// TIA Portal V17 export
// export: Created 2025-03-07T09:24:30.3982886Z, ExportSetting WithDefaults, DisplayName Totally Integrated Automation Portal, DisplayVersion V17 Update 8, DisplayName TIA Portal Openness, DisplayVersion V17 Update 8, DisplayName TIA Portal Version Control Interface, DisplayVersion V17, DisplayName SINAMICS Startdrive Advanced, DisplayVersion V17 SP2, DisplayName SINAMICS Startdrive G110M, G120, G120C, G120D, G120P, G115D, DisplayVersion V17 SP2, DisplayName SINAMICS Startdrive G130, G150, S120, S150, SINAMICS MV, S210, DisplayVersion V17 SP2, DisplayName STEP 7 Professional, DisplayVersion V17 Update 8, DisplayName SINUMERIK ONE STEP 7 Toolbox, DisplayVersion V17 Update 12, DisplayName SINUMERIK 840D sl STEP 7 Toolbox, DisplayVersion V17 Update 12, DisplayName STEP 7 Safety, DisplayVersion V17 Update 6, DisplayName WinCC Advanced, DisplayVersion V17 Update 8
FUNCTION "FC2202_PROFINET" : Void   // FC2202, LAD
{ S7_Optimized_Access := 'FALSE' }
AUTHOR : ETXETAR
VERSION : 1.0
// stored: AutoNumber false, IsIECCheckEnabled false, SetENOAutomatically false, UDAEnableTagReadback false
   VAR_TEMP
      COMMAND : Int;   // COMMAND
      BUSY : Bool;   // BUSY
   END_VAR
   VAR CONSTANT
      FC_NUMBER : Int := 2202;
   END_VAR
   VAR_TEMP   // added for the SCL form of the ladder/FBD networks
      _w1 : Bool;
   END_VAR
BEGIN

REGION Network 1: DEVICES STATES
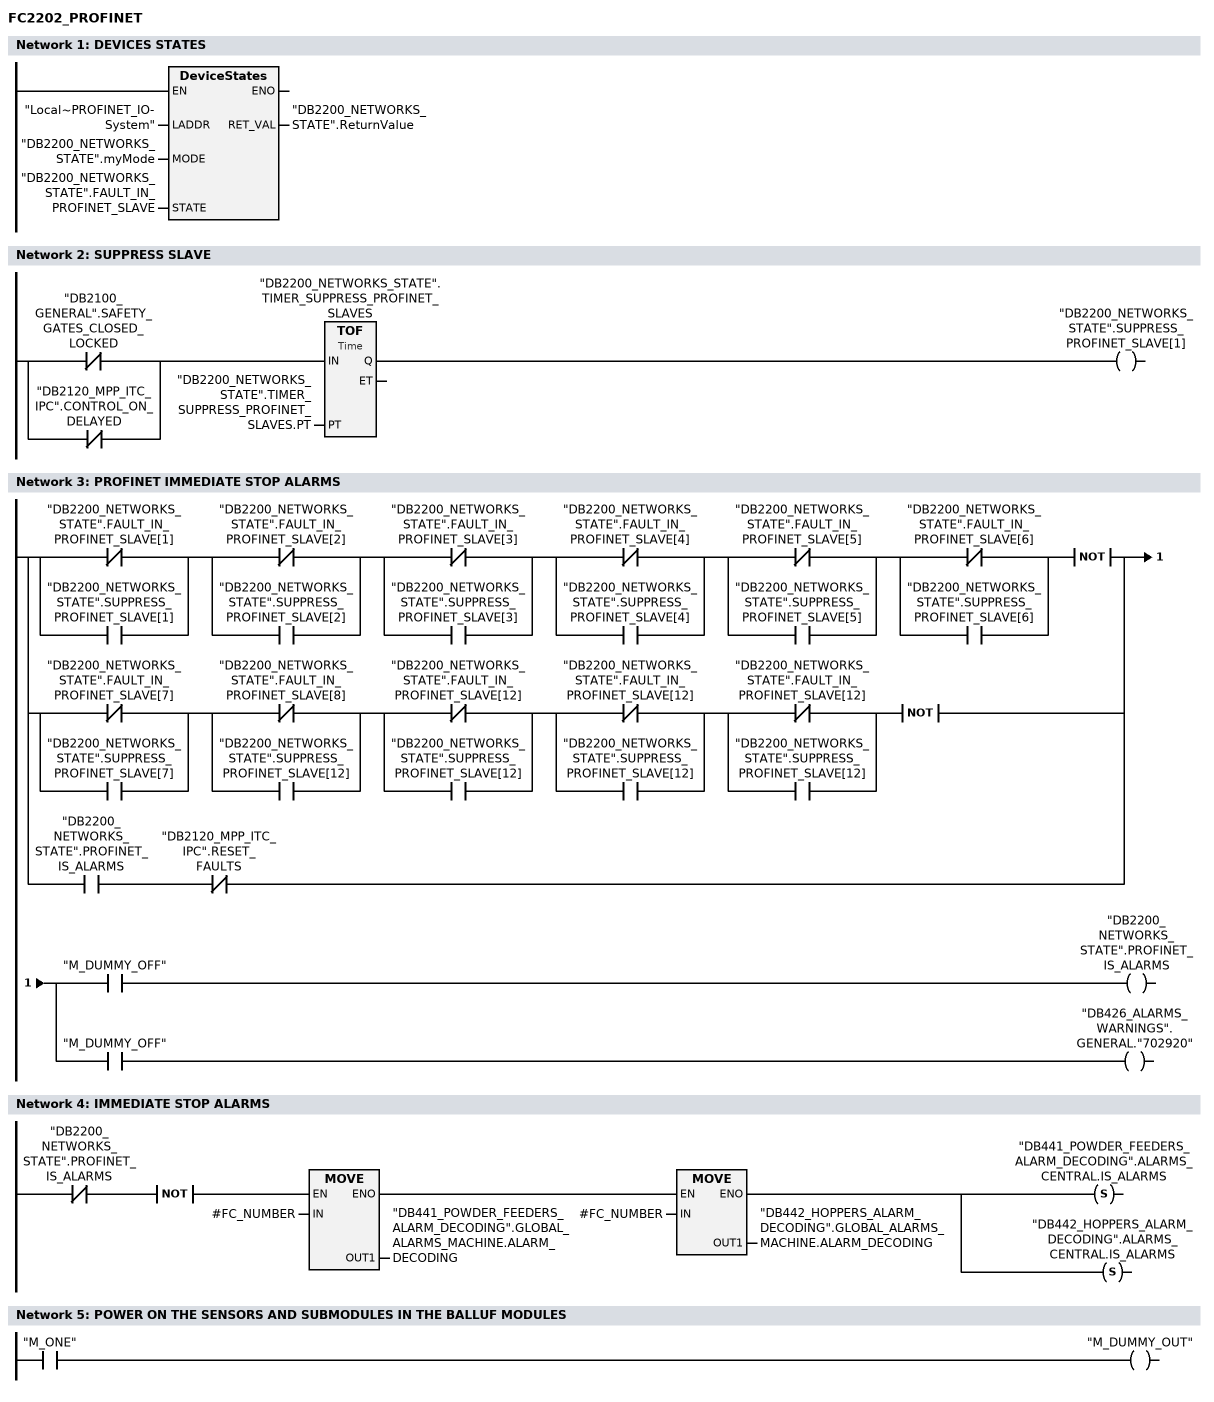
   RUNG wire#powerrail
      DeviceStates(LADDR := "Local~PROFINET_IO-System", MODE := "DB2200_NETWORKS_STATE".myMode, STATE := "DB2200_NETWORKS_STATE".FAULT_IN_PROFINET_SLAVE, Ret_Val => "DB2200_NETWORKS_STATE".ReturnValue)
   END_RUNG
   // the same network as SCL:
   "DB2200_NETWORKS_STATE".ReturnValue := DeviceStates(LADDR := "Local~PROFINET_IO-System",
                           MODE := "DB2200_NETWORKS_STATE".myMode,
                           STATE := "DB2200_NETWORKS_STATE".FAULT_IN_PROFINET_SLAVE);
END_REGION

REGION Network 2: SUPPRESS SLAVE
   RUNG wire#powerrail
      I_Contact( "DB2100_GENERAL".SAFETY_GATES_CLOSED_LOCKED )
      wire#w1
      { S7_Templates := "time_type := Time" } "DB2200_NETWORKS_STATE".TIMER_SUPPRESS_PROFINET_SLAVES.TOF(pt := "DB2200_NETWORKS_STATE".TIMER_SUPPRESS_PROFINET_SLAVES.PT, et =>)
      Coil( "DB2200_NETWORKS_STATE".SUPPRESS_PROFINET_SLAVE[1] )
   END_RUNG
   RUNG wire#powerrail
      I_Contact( "DB2120_MPP_ITC_IPC".CONTROL_ON_DELAYED )
   END_RUNG wire#w1
   // the same network as SCL:
   "DB2200_NETWORKS_STATE".TIMER_SUPPRESS_PROFINET_SLAVES.TOF(IN := NOT "DB2100_GENERAL".SAFETY_GATES_CLOSED_LOCKED OR NOT "DB2120_MPP_ITC_IPC".CONTROL_ON_DELAYED,
                           PT := "DB2200_NETWORKS_STATE".TIMER_SUPPRESS_PROFINET_SLAVES.PT);
   "DB2200_NETWORKS_STATE".SUPPRESS_PROFINET_SLAVE[1] := "DB2200_NETWORKS_STATE".TIMER_SUPPRESS_PROFINET_SLAVES.Q;
END_REGION

REGION Network 3: PROFINET IMMEDIATE STOP ALARMS
   RUNG wire#powerrail
      I_Contact( "DB2200_NETWORKS_STATE".FAULT_IN_PROFINET_SLAVE[1] )
      wire#w1
      I_Contact( "DB2200_NETWORKS_STATE".FAULT_IN_PROFINET_SLAVE[2] )
      wire#w2
      I_Contact( "DB2200_NETWORKS_STATE".FAULT_IN_PROFINET_SLAVE[3] )
      wire#w3
      I_Contact( "DB2200_NETWORKS_STATE".FAULT_IN_PROFINET_SLAVE[4] )
      wire#w4
      I_Contact( "DB2200_NETWORKS_STATE".FAULT_IN_PROFINET_SLAVE[5] )
      wire#w5
      I_Contact( "DB2200_NETWORKS_STATE".FAULT_IN_PROFINET_SLAVE[6] )
      wire#w6
      Not()
      wire#w7
      Contact( "M_DUMMY_OFF" )
      Coil( "DB2200_NETWORKS_STATE".PROFINET_IS_ALARMS )
   END_RUNG
   RUNG wire#powerrail
      Contact( "DB2200_NETWORKS_STATE".SUPPRESS_PROFINET_SLAVE[1] )
   END_RUNG wire#w1
   RUNG wire#w1
      Contact( "DB2200_NETWORKS_STATE".SUPPRESS_PROFINET_SLAVE[2] )
   END_RUNG wire#w2
   RUNG wire#w2
      Contact( "DB2200_NETWORKS_STATE".SUPPRESS_PROFINET_SLAVE[3] )
   END_RUNG wire#w3
   RUNG wire#w3
      Contact( "DB2200_NETWORKS_STATE".SUPPRESS_PROFINET_SLAVE[4] )
   END_RUNG wire#w4
   RUNG wire#w4
      Contact( "DB2200_NETWORKS_STATE".SUPPRESS_PROFINET_SLAVE[5] )
   END_RUNG wire#w5
   RUNG wire#w5
      Contact( "DB2200_NETWORKS_STATE".SUPPRESS_PROFINET_SLAVE[6] )
   END_RUNG wire#w6
   RUNG wire#powerrail
      I_Contact( "DB2200_NETWORKS_STATE".FAULT_IN_PROFINET_SLAVE[7] )
      wire#w8
      I_Contact( "DB2200_NETWORKS_STATE".FAULT_IN_PROFINET_SLAVE[8] )
      wire#w9
      I_Contact( "DB2200_NETWORKS_STATE".FAULT_IN_PROFINET_SLAVE[12] )
      wire#w10
      I_Contact( "DB2200_NETWORKS_STATE".FAULT_IN_PROFINET_SLAVE[12] )
      wire#w11
      I_Contact( "DB2200_NETWORKS_STATE".FAULT_IN_PROFINET_SLAVE[12] )
      wire#w12
      Not()
   END_RUNG wire#w7
   RUNG wire#powerrail
      Contact( "DB2200_NETWORKS_STATE".SUPPRESS_PROFINET_SLAVE[7] )
   END_RUNG wire#w8
   RUNG wire#w8
      Contact( "DB2200_NETWORKS_STATE".SUPPRESS_PROFINET_SLAVE[12] )
   END_RUNG wire#w9
   RUNG wire#w9
      Contact( "DB2200_NETWORKS_STATE".SUPPRESS_PROFINET_SLAVE[12] )
   END_RUNG wire#w10
   RUNG wire#w10
      Contact( "DB2200_NETWORKS_STATE".SUPPRESS_PROFINET_SLAVE[12] )
   END_RUNG wire#w11
   RUNG wire#w11
      Contact( "DB2200_NETWORKS_STATE".SUPPRESS_PROFINET_SLAVE[12] )
   END_RUNG wire#w12
   RUNG wire#powerrail
      Contact( "DB2200_NETWORKS_STATE".PROFINET_IS_ALARMS )
      I_Contact( "DB2120_MPP_ITC_IPC".RESET_FAULTS )
   END_RUNG wire#w7
   RUNG wire#w7
      Contact( "M_DUMMY_OFF" )
      Coil( "DB426_ALARMS_WARNINGS".GENERAL."702920" )
   END_RUNG
   // the same network as SCL:
   #_w1 := NOT ((NOT "DB2200_NETWORKS_STATE".FAULT_IN_PROFINET_SLAVE[1] OR "DB2200_NETWORKS_STATE".SUPPRESS_PROFINET_SLAVE[1]) AND (NOT "DB2200_NETWORKS_STATE".FAULT_IN_PROFINET_SLAVE[2] OR "DB2200_NETWORKS_STATE".SUPPRESS_PROFINET_SLAVE[2]) AND (NOT "DB2200_NETWORKS_STATE".FAULT_IN_PROFINET_SLAVE[3] OR "DB2200_NETWORKS_STATE".SUPPRESS_PROFINET_SLAVE[3]) AND (NOT "DB2200_NETWORKS_STATE".FAULT_IN_PROFINET_SLAVE[4] OR "DB2200_NETWORKS_STATE".SUPPRESS_PROFINET_SLAVE[4]) AND (NOT "DB2200_NETWORKS_STATE".FAULT_IN_PROFINET_SLAVE[5] OR "DB2200_NETWORKS_STATE".SUPPRESS_PROFINET_SLAVE[5]) AND (NOT "DB2200_NETWORKS_STATE".FAULT_IN_PROFINET_SLAVE[6] OR "DB2200_NETWORKS_STATE".SUPPRESS_PROFINET_SLAVE[6])) OR NOT ((NOT "DB2200_NETWORKS_STATE".FAULT_IN_PROFINET_SLAVE[7] OR "DB2200_NETWORKS_STATE".SUPPRESS_PROFINET_SLAVE[7]) AND (NOT "DB2200_NETWORKS_STATE".FAULT_IN_PROFINET_SLAVE[8] OR "DB2200_NETWORKS_STATE".SUPPRESS_PROFINET_SLAVE[12]) AND (NOT "DB2200_NETWORKS_STATE".FAULT_IN_PROFINET_SLAVE[12] OR "DB2200_NETWORKS_STATE".SUPPRESS_PROFINET_SLAVE[12]) AND (NOT "DB2200_NETWORKS_STATE".FAULT_IN_PROFINET_SLAVE[12] OR "DB2200_NETWORKS_STATE".SUPPRESS_PROFINET_SLAVE[12]) AND (NOT "DB2200_NETWORKS_STATE".FAULT_IN_PROFINET_SLAVE[12] OR "DB2200_NETWORKS_STATE".SUPPRESS_PROFINET_SLAVE[12])) OR ("DB2200_NETWORKS_STATE".PROFINET_IS_ALARMS AND NOT "DB2120_MPP_ITC_IPC".RESET_FAULTS);
   "DB2200_NETWORKS_STATE".PROFINET_IS_ALARMS := #_w1 AND "M_DUMMY_OFF";
   "DB426_ALARMS_WARNINGS".GENERAL."702920" := #_w1 AND "M_DUMMY_OFF";
END_REGION

REGION Network 4: IMMEDIATE STOP ALARMS
   RUNG wire#powerrail
      I_Contact( "DB2200_NETWORKS_STATE".PROFINET_IS_ALARMS )
      Not()
      { S7_GenerateENO := "TRUE" } Move(in := #FC_NUMBER, out1 => "DB441_POWDER_FEEDERS_ALARM_DECODING".GLOBAL_ALARMS_MACHINE.ALARM_DECODING)
      { S7_GenerateENO := "TRUE" } Move(in := #FC_NUMBER, out1 => "DB442_HOPPERS_ALARM_DECODING".GLOBAL_ALARMS_MACHINE.ALARM_DECODING)
      wire#w1
      S_Coil( "DB441_POWDER_FEEDERS_ALARM_DECODING".ALARMS_CENTRAL.IS_ALARMS )
   END_RUNG
   RUNG wire#w1
      S_Coil( "DB442_HOPPERS_ALARM_DECODING".ALARMS_CENTRAL.IS_ALARMS )
   END_RUNG
   // the same network as SCL:
   // ENO of a box is taken as its EN; it also drops when the box reports an error
   IF NOT (NOT "DB2200_NETWORKS_STATE".PROFINET_IS_ALARMS) THEN
       "DB441_POWDER_FEEDERS_ALARM_DECODING".GLOBAL_ALARMS_MACHINE.ALARM_DECODING := #FC_NUMBER;
       "DB442_HOPPERS_ALARM_DECODING".GLOBAL_ALARMS_MACHINE.ALARM_DECODING := #FC_NUMBER;
       "DB441_POWDER_FEEDERS_ALARM_DECODING".ALARMS_CENTRAL.IS_ALARMS := TRUE;
       "DB442_HOPPERS_ALARM_DECODING".ALARMS_CENTRAL.IS_ALARMS := TRUE;
   END_IF;
END_REGION

REGION Network 5: POWER ON THE SENSORS AND SUBMODULES IN THE BALLUF MODULES
   RUNG wire#powerrail
      Contact( "M_ONE" )
      Coil( "M_DUMMY_OUT" )
   END_RUNG
   // the same network as SCL:
   "M_DUMMY_OUT" := "M_ONE";
END_REGION
END_FUNCTION
